(* IEC 61131-3 sources: router_agent/data/raw-data/benchmark_raw/215_SelectSort/plc_st_files, 1 file *)

(* ---- 215_SelectSort.st ---- *)
FUNCTION_BLOCK SelectSort
VAR_INPUT
    exe : BOOL;
    seq : ARRAY[1..10] OF LREAL;
END_VAR

VAR_OUTPUT
    error : BOOL;
    status : WORD;
END_VAR

VAR
    i, j, min_idx : INT;
    temp : LREAL;
    arr_len : INT := 5;
END_VAR

IF exe THEN
    FOR i := 1 TO arr_len - 1 DO
        min_idx := i;
        FOR j := i + 1 TO arr_len DO
            IF seq[j] < seq[min_idx] THEN
                min_idx := j;
            END_IF;
        END_FOR;

        IF min_idx <> i THEN
            temp := seq[i];
            seq[i] := seq[min_idx];
            seq[min_idx] := temp;
        END_IF;
    END_FOR;

    error := FALSE;
    status := 16#0000;

END_IF;
END_FUNCTION_BLOCK
